(* IEC 61131-3 sources: SRCI/RobotLibrary/RobotLibrary/POUs/Spline/MC_CreateSpline, 1 file *)

(* ---- MC_CreateSplineFB.st ---- *)
/// Create spline on RC from positions stored in PLC
FUNCTION_BLOCK MC_CreateSplineFB EXTENDS RobotLibraryBaseExecuteFB
// -------------------------------------------------------------------------
//  SRCI Robot Library
// -------------------------------------------------------------------------
//
//  Object:      CreateSplineFB
//  Author:      Thorsten Brach
//  Date:        2024-06-01
//
//  Description:
//
//
//  Copyright:
//    (C) 2024 Thorsten Brach. All rights reserved
//             Licensed under the LGPL-3.0 license.
//
//  Disclaimer:
//    This project is provided without any guarantee and can be used for
//    private and commercial purposes. Any use is at the user’s
//    own risk and responsibility.
//
// -------------------------------------------------------------------------
VAR_INPUT
  /// command parameter
  ParCmd          : CreateSplineParCmd;
END_VAR
VAR_OUTPUT
  /// Command is transferred and confirmed by the RC
  CommandBuffered : BOOL;
  /// command results
  OutCmd          : CreateSplineOutCmd;
END_VAR

VAR
  /// internal copy of command parameter
 _parCmd          : CreateSplineParCmd;
  /// command data to send
 _command         : CreateSplineSendData;
  /// response data received
 _response        : CreateSplineRecvData;
END_VAR

  SUPER^(AxesGroup := AxesGroup);

END_FUNCTION_BLOCK

METHOD CheckParameterChanged : BOOL
VAR_IN_OUT
  /// Robot assignment of function
  AxesGroup    : AxesGroup;
END_VAR

  // Check ParCmd Size is > 0, becaue MemCmp does not work correctly with size = 0
  IF (SIZEOF(ParCmd) = 0)
  THEN
    RETURN;
  END_IF

  // compare memory
  CheckParameterChanged := ( MemCmp(ADR(ParCmd), ADR(_parCmd), SIZEOF(ParCmd)) <> RobotLibraryConstants.OK );

  IF ( CheckParameterChanged )
  THEN
    // update internal copy of parameters
   _parCmd := ParCmd;
    // inc parameter sequence
   _command.ParSeq := _command.ParSeq + 1;
    // update command data
    CommandData := CreateCommandPayload(); // ( Access via reference to rCommandFB in ACR )
    // notify active command register
    AxesGroup.Acyclic.ActiveCommandRegister.NotifyParameterChanged := _uniqueID;
  END_IF

END_METHOD

METHOD INTERNAL CreateCommandPayload : SendData
// Table 6-754: Sent CMD payload (PLC to RC) of "CreateSpline"
// --------------------------
// Header
// --------------------------
// Byte 00 : UINT  - Type HB
// Byte 01 :       - Type LB
// Byte 02 : USINT - Reserve | ExecutionMode
// Byte 03 : USINT - ParSeq  | Priority
// --------------------------
// Datablock
// --------------------------
// Byte 04 : UINT  Mode;
// Byte 05 : SINT  SplineID;
// Byte 06 : UINT  SplineData.VelocityRate;
// Byte 07 :       SplineData.VelocityRate;
// Byte 08 : UINT  SplineData.AccelerationRate;
// Byte 09 :       SplineData.AccelerationRate;
// Byte 10 : UINT  SplineData.DecelerationRate;
// Byte 11 :       SplineData.DecelerationRate;
// Byte 12 : UINT  SplineData.JerkRate;
// Byte 13 :       SplineData.JerkRate;
// Byte 14 : USINT SplineData.ToolNo;
// Byte 15 : USINT SplineData.FrameNo;
// Byte 16 : REAL  SplineData.X;
// Byte 17 :       SplineData.X;
// Byte 18 :       SplineData.X;
// Byte 19 :       SplineData.X;
// Byte 20 : REAL  SplineData.Y;
// Byte 21 :       SplineData.Y;
// Byte 22 :       SplineData.Y;
// Byte 23 :       SplineData.Y;
// Byte 24 : REAL  SplineData.Z;
// Byte 25 :       SplineData.Z;
// Byte 26 :       SplineData.Z;
// Byte 27 :       SplineData.Z;
// Byte 28 : REAL  SplineData.RX;
// Byte 29 :       SplineData.RX;
// Byte 30 :       SplineData.RX;
// Byte 31 :       SplineData.RX;
// Byte 32 : REAL  SplineData.RY;
// Byte 33 :       SplineData.RY;
// Byte 34 :       SplineData.RY;
// Byte 35 :       SplineData.RY;
// Byte 36 : REAL  SplineData.RZ;
// Byte 37 :       SplineData.RZ;
// Byte 38 :       SplineData.RZ;
// Byte 39 :       SplineData.RZ;
// Byte 40 : BYTE  - - - - - W E S;
// Byte 41 : BYTE  Reserved;
// Byte 42 : BYTE  SplineData.TurnNumber[0];
// Byte 43 : BYTE  SplineData.TurnNumber[1];
// Byte 44 : BYTE  SplineData.TurnNumber[2];
// Byte 45 : BYTE  SplineData.TurnNumber[3];
// Byte 46 : REAL  SplineData.E1;
// Byte 47 :       SplineData.E1;
// Byte 48 :       SplineData.E1;
// Byte 49 :       SplineData.E1;
// Byte 50 : UINT  SplineData.Time;
// Byte 51 :       SplineData.Time;
// Byte 52 : REAL  SplineData.E2;
// Byte 53 :       SplineData.E2;
// Byte 54 :       SplineData.E2;
// Byte 55 :       SplineData.E2;
// Byte 56 : REAL  SplineData.E3;
// Byte 57 :       SplineData.E3;
// Byte 58 :       SplineData.E3;
// Byte 59 :       SplineData.E3;
// Byte 60 : REAL  SplineData.E4;
// Byte 61 :       SplineData.E4;
// Byte 62 :       SplineData.E4;
// Byte 63 :       SplineData.E4;
// Byte 64 : REAL  SplineData.E5;
// Byte 65 :       SplineData.E5;
// Byte 66 :       SplineData.E5;
// Byte 67 :       SplineData.E5;
// Byte 68 : REAL  SplineData.E6;
// Byte 69 :       SplineData.E6;
// Byte 70 :       SplineData.E6;
// Byte 71 :       SplineData.E6;
VAR
  /// internal index for loops
  _idx : DINT;
END_VAR

  // set command parameter
  _command.CmdTyp   :=  CmdType.CreateSpline;
  _command.ExecMode :=  ExecMode;
  _command.ParSeq   := _command.ParSeq;
  _command.Priority :=  Priority;
  _command.Mode     := _parCmd.Mode;
  _command.SplineID := _parCmd.SplineID;

  FOR _idx := 1 TO RobotLibraryParameter.SPLINE_DATA_MAX
  DO
    _command.SplineData[_idx].VelocityRate     := REAL_TO_UINT(_parCmd.SplineData[_idx].VelocityRate     * RobotLibraryConstants.REAL_CONVERSION_FACTOR);
    _command.SplineData[_idx].AccelerationRate := REAL_TO_UINT(_parCmd.SplineData[_idx].AccelerationRate * RobotLibraryConstants.REAL_CONVERSION_FACTOR);
    _command.SplineData[_idx].DecelerationRate := REAL_TO_UINT(_parCmd.SplineData[_idx].DecelerationRate * RobotLibraryConstants.REAL_CONVERSION_FACTOR);
    _command.SplineData[_idx].JerkRate         := REAL_TO_UINT(_parCmd.SplineData[_idx].JerkRate         * RobotLibraryConstants.REAL_CONVERSION_FACTOR);
    _command.SplineData[_idx].ToolNo           :=              _parCmd.SplineData[_idx].ToolNo;
    _command.SplineData[_idx].FrameNo          :=              _parCmd.SplineData[_idx].FrameNo;
    _command.SplineData[_idx].MoveTime         := TIME_TO_UINT(_parCmd.SplineData[_idx].MoveTime);
  END_FOR

  // copy command data to header
  _cmdHeader := _command;
  // call base implementation to copy header to payload buffer
  CreateCommandPayload := SUPER^.CreateCommandPayload();

  // add command.Mode
  CreateCommandPayload.AddUint(_command.Mode);
  // add command.SplineID
  CreateCommandPayload.AddSint(_command.SplineID);

  FOR _idx := 1 TO RobotLibraryParameter.SPLINE_DATA_MAX
  DO
    // add command.VelocityRate
    CreateCommandPayload.AddUint(_command.SplineData[_idx].VelocityRate);
    // add command.AccelerationRate
    CreateCommandPayload.AddUint(_command.SplineData[_idx].AccelerationRate);
    // add command.DecelerationRate
    CreateCommandPayload.AddUint(_command.SplineData[_idx].DecelerationRate);
    // add command.JerkRate
    CreateCommandPayload.AddUint(_command.SplineData[_idx].JerkRate);
    // add command.ToolNo
    CreateCommandPayload.AddUsint(_command.SplineData[_idx].ToolNo);
    // add command.FrameNo
    CreateCommandPayload.AddUsint(_command.SplineData[_idx].FrameNo);
    // add command.SplineData[_idx].Position.X
    CreateCommandPayload.AddReal(_command.SplineData[_idx].Position.X);
    // add command.SplineData[_idx].Position.Y
    CreateCommandPayload.AddReal(_command.SplineData[_idx].Position.Y);
    // add command.SplineData[_idx].Position.Z
    CreateCommandPayload.AddReal(_command.SplineData[_idx].Position.Z);
    // add command.SplineData[_idx].Position.Rx
    CreateCommandPayload.AddReal(_command.SplineData[_idx].Position.Rx);
    // add command.SplineData[_idx].Position.Ry
    CreateCommandPayload.AddReal(_command.SplineData[_idx].Position.Ry);
    // add command.SplineData[_idx].Position.Rz
    CreateCommandPayload.AddReal(_command.SplineData[_idx].Position.Rz);
    // add command.SplineData[_idx].Position.Config
    CreateCommandPayload.AddArmConfig(_command.SplineData[_idx].Position.Config);
    // add command.SplineData[_idx].Position.TurnNumber
    CreateCommandPayload.AddTurnNumber(_command.SplineData[_idx].Position.TurnNumber);
    // add command.SplineData[_idx].Position.E1
    CreateCommandPayload.AddReal(_command.SplineData[_idx].Position.E1);
    // add command.SplineData[_idx].MoveTime
    CreateCommandPayload.AddUint(_command.SplineData[_idx].MoveTime);
    // add command.SplineData[_idx].Position.E2
    CreateCommandPayload.AddReal(_command.SplineData[_idx].Position.E2);
    // add command.SplineData[_idx].Position.E3
    CreateCommandPayload.AddReal(_command.SplineData[_idx].Position.E3);
    // add command.SplineData[_idx].Position.E4
    CreateCommandPayload.AddReal(_command.SplineData[_idx].Position.E4);
    // add command.SplineData[_idx].Position.E5
    CreateCommandPayload.AddReal(_command.SplineData[_idx].Position.E5);
    // add command.SplineData[_idx].Position.E6
    CreateCommandPayload.AddReal(_command.SplineData[_idx].Position.E6);
  END_FOR

END_METHOD

METHOD FB_init : BOOL
VAR_INPUT
  /// if TRUE, the retain variables are initialized (warm start / cold start)
	bInitRetains : BOOL;
  /// if TRUE, the instance afterwards gets moved into the copy code (online change)
	bInCopyCode  : BOOL;
END_VAR

  MyType := 'MC_CreateSplineFB';

  ExecMode := ExecutionMode.PARALLEL;

END_METHOD

METHOD PROTECTED OnCall
VAR_IN_OUT
  /// Robot assignment of function
  AxesGroup : AxesGroup;
END_VAR

  // call base implementation
  SUPER^.OnCall(AxesGroup := AxesGroup);

  CASE _stepCmd OF

    00:  IF ( _execute_R.Q )
         THEN
           // set busy flag
           Busy := TRUE;
           // Reset command outputs
           MemSet(ADR(OutCmd),0,SIZEOF(OutCmd));
           // apply command parameter
          _parCmd := ParCmd;
           // init parameter sequence
          _command.ParSeq := 1;
           // set timeout
           SetTimeout(PT := _timeoutCmd, rTimer := _timerCmd);
           // inc step counter
          _stepCmd := _stepCmd + 1;
  	     END_IF

    01:  // create command data
         CommandData := CreateCommandPayload();
         // Add command to active command register
        _uniqueID := AxesGroup.Acyclic.ActiveCommandRegister.AddCmd( pCommandFB := ADR(THIS^ ));
         // set timeout
         SetTimeout(PT := _timeoutCmd, rTimer := _timerCmd);
         // inc step counter
        _stepCmd := _stepCmd + 1;

    02:  // Wait for responce received
         IF ( _responseReceived )
         THEN
           // reset response received flag
          _responseReceived := FALSE;

           CASE  _response.State
           OF
             CmdMessageState.BUFFERED : CommandBuffered := TRUE;
             CmdMessageState.DONE     : Done            := TRUE;
             CmdMessageState.ERROR    : Error           := TRUE;
  				 END_CASE

           // Done, Aborted or Error ?
           IF (_response.State >= CmdMessageState.DONE )
           THEN
             // Reset Busy flag
             Busy := FALSE;
             // set timeout
             SetTimeout(PT := _timeoutCmd, rTimer := _timerCmd);
             // inc step counter
            _stepCmd := _stepCmd + 1;
  				 END_IF
         END_IF

    03: IF ( NOT Execute)
        THEN
          Reset();
  			END_IF
  ELSE
    // invalid step
    ErrorID := RobotLibraryEvents.ERR_INVALID_STEP;
  END_CASE

  // Cancel
  IF (Busy) AND (NOT Execute)
  THEN
    // try to remove cmd
    AxesGroup.Acyclic.ActiveCommandRegister.RemoveCmd(_uniqueID);
  END_IF

  // Reset FB
  IF ( NOT Execute )
  THEN
    Reset();
  END_IF

END_METHOD

METHOD INTERNAL ParseResponsePayload : DINT
// Table 6-755: Received CMD payload (RC to PLC) of "CreateSpline"
// --------------------------
// Header
// --------------------------
// Byte 00 : USINT   - ParSeq | State
// Byte 01 : SINT    - AlarmMessageSeverity
// Byte 02 : UINT    - AlarmMessageCode HB
// Byte 03 :         - AlarmMessageCode LB
VAR_INPUT
  /// Response data
  ResponseData : RecvData;
END_VAR

  // call base implementation to parse the header from payload buffer
  ResponseData.PayloadPtr := SUPER^.ParseResponsePayload(ResponseData);

  // copy parsed header to response
  _response.ParSeq               := _rspHeader.ParSeq;
  _response.State                := _rspHeader.State;
  _response.AlarmMessageSeverity := _rspHeader.AlarmMessageSeverity;
  _response.AlarmMessageCode     := _rspHeader.AlarmMessageCode;

END_METHOD

METHOD PROTECTED Reset : DINT
VAR_INPUT
END_VAR

  Reset := SUPER^.Reset();

  Done               := FALSE;
  Busy               := FALSE;
  CommandBuffered    := FALSE;

END_METHOD
